FUNCTION_BLOCK ABSTRACT Crane_MoveBase EXTENDS ControlPrimitiveBase
VAR_INPUT
END_VAR
VAR_OUTPUT
END_VAR
VAR
	m_ptrCrane: POINTER TO Crane;
END_VAR

SUPER^();

METHOD Abort : BOOL
VAR_INPUT
END_VAR
m_ptrCrane^.METH_CarrierStop();
Abort := TRUE;
END_METHOD

PROPERTY ABSTRACT AtTarget : BOOL
GET
END_GET
END_PROPERTY

(* Execution logic of this Control Primitive. *)
METHOD PROTECTED ExecuteInternal : BOOL
VAR_INPUT
	i_params	: Resi4MPM.ParameterSet;
END_VAR
VAR
	angle: REAL;
	diff: REAL;
END_VAR
angle := m_st^.GetNumeric(EProcessVariables.Crane_Angle);
diff := TargetAngle - angle;

IF AtTarget THEN
	m_ptrCrane^.METH_CarrierStop();
	ExecuteInternal := TRUE;
ELSIF diff < 0 THEN
	m_ptrCrane^.METH_CarrierTurnClockwise();
ELSE
	m_ptrCrane^.METH_CarrierTurnCounterClockwise();
END_IF
END_METHOD

PROPERTY ABSTRACT TargetAngle : UINT
GET
END_GET
END_PROPERTY

END_FUNCTION_BLOCK

(* stored: Version 1.1.0.1
   POU Crane_MoveBase: Id {3b3ba2fc-ae22-4a3d-905d-30807d575792}, SpecialFunc None
   Method Abort: Id {24c43fc6-d168-4705-bfa5-21f2596b0748}
   Property AtTarget: Id {7d293d69-b76c-46b2-a173-ca6dfc2465b7}
   Get Get: Id {ebf3003d-70ed-464d-964b-52a16a3efc17}
   Method ExecuteInternal: Id {717bfc26-f876-4ff8-abc2-bfb1b933bc98}
   Property TargetAngle: Id {c39d77f4-a728-45f6-bf29-f72c6181dc14}
   Get Get: Id {16fd91db-7002-4ae9-85a7-017d501b8296} *)
